# EPICS autosave request: tomoScanApp/Db/tomoScan_19BM_settings.req
# This file is used by autosave to determine what PVs to save
# It is also used by tomoScan to determine what PVs to create

# This is the file for the tomoscan_19bm derived class.
# It matches tomoScan_7BM_settings.req with the gain-field entries removed.

####################
# Energy information
####################
$(P)$(R)Energy
$(P)$(R)EnergyMode

#########################
# Beam status information
#########################
$(P)$(R)BeamReadyPVName
$(P)$(R)BeamReadyValue
$(P)$(R)Testing

################
# Shutter status
################
$(P)$(R)ShutterStatusPVName

####################
# Optics information
####################
$(P)$(R)ScintillatorType
$(P)$(R)ScintillatorThickness
$(P)$(R)ImagePixelSize
$(P)$(R)DetectorPixelSize
$(P)$(R)CameraObjective
$(P)$(R)CameraTubeLength
$(P)$(R)CameraDistance

####################
# Sample information
####################
$(P)$(R)SampleName
$(P)$(R)SampleDescription1
$(P)$(R)SampleDescription2
$(P)$(R)SampleDescription3

##################
# User information
##################
$(P)$(R)UserName
$(P)$(R)UserInstitution
$(P)$(R)UserBadge
$(P)$(R)UserEmail
$(P)$(R)ProposalNumber
$(P)$(R)ProposalTitle
$(P)$(R)ESAFNumber
$(P)$(R)UserInfoUpdate

#################
# Data management
#################
$(P)$(R)DetectorTopDir
$(P)$(R)UserLastName
$(P)$(R)ExperimentYearMonth
$(P)$(R)RemoteAnalysisDir
$(P)$(R)CopyToAnalysisDir

#########################
# Camera External Trigger
#########################
$(P)$(R)ExternalTriggerSource
